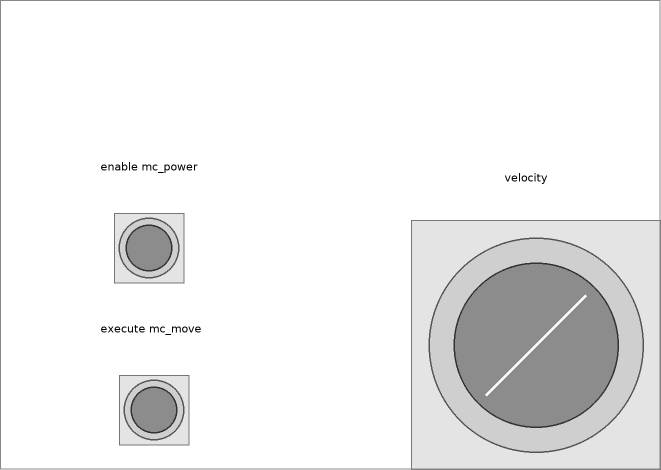
VISUALIZATION Visualization  // 661x470
    PushSwitchLed (114,213 70x70), variable: MAIN.bEnable, behaviour: TOGGLE, style: Switch-PushSwitchLed-Gray
    PushSwitchLed (119,375 70x70), variable: MAIN.bExecute, behaviour: TOGGLE, style: Switch-PushSwitchLed-Gray
    Label (74,152 150x30), "enable mc_power"
    Label (76,314 150x30), "execute mc_move"
    Potentiometer360 (411,220 250x250), variable: MAIN.rVelocity, style: Potentiometer-Potentiometer360-Gray, scale format: %.1f, scale 0..5000
        p2431819421: Outside
    Label (451,163 150x30), "velocity"
END_VISUALIZATION

(* stored: Version 1.1.0.1, ProductVersion 3.1.4024.9
   Visu Visualization: Id {9bcfcc5d-8f60-4754-a1b1-94fe0e97b05f} *)
